TYPE E_PulsGen :
(**************************************************************************************
 * 	Application		:	BoxControl Framework
 *	Revision		:	$Revision: 404529 $
 *	Revision date	:	$Date: 2018-04-23 08:21:38 +0200 (Mo., 23 Apr 2018) $
 *	Last changed by	:	$Author: b7bolm $
 *	URL				:	$URL: http://almscdc.swisslog.com/repo/SWPD/Development/BoxControlFramework/20_Release/trunk/01_Software/BCF/BCF/JumpStart/30_Toolbox/13_TimerCounter/01_DUTs/E_PulsGen.TcDUT $
 *
 *	Purpose			:	Pulse generator
 *
 * ------------------------------------------------------------------------------------
 *	Copyright Swisslog [IP AG], Switzerland. All rights reserved.
 * 
 * ------------------------------------------------------------------------------------
 *	
 * 	Revision History: 
 *
 * 	VERSION			DATE			INITIALS			DESCRIPTION
 *	0.1				01.01.2001		swl					Example
 *
 **************************************************************************************)
(
	PG_READY,
	PG_BUSY,
	PG_END
);
END_TYPE

(* stored: Version 1.1.0.1, ProductVersion 3.1.4020.6
   DUT E_PulsGen: Id {ba2381f0-f74c-4e73-8f3b-894c439f74bd} *)
